FUNCTION_BLOCK EulerAngleOrientation EXTENDS AngleSequenceOrientation
VAR_INPUT
END_VAR
VAR_OUTPUT
END_VAR
VAR
	Angles_ : ARRAY [0..2] OF LREAL; 
	Sequence_ : EulerAngleSequence;
END_VAR

METHOD PUBLIC Clear
VAR_INPUT
END_VAR
Angles_[0] := 0;
Angles_[1] := 0;
Angles_[2] := 0;
END_METHOD

METHOD PUBLIC CopyFrom
VAR_INPUT
	O : EulerAngleOrientation;
END_VAR
CLEAR();
Sequence := O.Sequence;
AngleAccessor.CopyFrom(O.AngleAccessor);
END_METHOD

METHOD PUBLIC  GetAngle : LREAL
VAR_INPUT
	I : UINT;
END_VAR
VAR
	Angles : ARRAY [0..2] OF LREAL;
END_VAR
IF I >= Length THEN
	GetAngle := 0;
	RETURN;
END_IF

GetAngle := Angles[I];
END_METHOD

METHOD PUBLIC  GetDimension : Dimension
VAR_INPUT
	I : UINT;
END_VAR
VAR
	Dims : ARRAY [0..2] OF Dimension;
END_VAR
IF I >= Length THEN
	GetDimension := 0;
	RETURN;
END_IF

Dims := GetDimensions();
GetDimension := Dims[I];
END_METHOD

METHOD PUBLIC GetDimensions : ARRAY [0..2] OF Dimension
VAR_INPUT
END_VAR
CASE Sequence OF
	EulerAngleSequence.XYX:
		GetDimensions[0] := 0;
		GetDimensions[1] := 1;
		GetDimensions[2] := 0;
	EulerAngleSequence.XZX:
		GetDimensions[0] := 0;
		GetDimensions[1] := 2;
		GetDimensions[2] := 0;
	EulerAngleSequence.YXY:
		GetDimensions[0] := 1;
		GetDimensions[1] := 0;
		GetDimensions[2] := 1;
	EulerAngleSequence.YZY:
		GetDimensions[0] := 1;
		GetDimensions[1] := 2;
		GetDimensions[2] := 1;
	EulerAngleSequence.ZXZ:
		GetDimensions[0] := 2;
		GetDimensions[1] := 0;
		GetDimensions[2] := 2;
	EulerAngleSequence.ZYZ:
		GetDimensions[0] := 2;
		GetDimensions[1] := 1;
		GetDimensions[2] := 2;
	ELSE
		GetDimensions[0] := 0;
		GetDimensions[1] := 0;
		GetDimensions[2] := 0;
END_CASE
END_METHOD

PROPERTY Length : UINT
GET
Length := 3;
END_GET
END_PROPERTY

PROPERTY PUBLIC RaDeg : LREAL
GET
RaDeg := 180 * Angles_[0] / PI;
END_GET
SET
Angles_[0] := PI * RaDeg / 180;
END_SET
END_PROPERTY

PROPERTY PUBLIC RaRad : LREAL
GET
RaRad := Angles_[0];
END_GET
SET
Angles_[0] := RaRad;
END_SET
END_PROPERTY

PROPERTY PUBLIC RbDeg : LREAL
GET
RbDeg := 180 * Angles_[1] / PI;
END_GET
SET
Angles_[1] := PI * RbDeg / 180;
END_SET
END_PROPERTY

PROPERTY PUBLIC RbRad : LREAL
GET
RbRad := Angles_[1];
END_GET
SET
Angles_[1] := RbRad;
END_SET
END_PROPERTY

PROPERTY PUBLIC RcDeg : LREAL
GET
RcDeg := 180 * Angles_[2] / PI;
END_GET
SET
Angles_[2] := PI * RcDeg / 180;
END_SET
END_PROPERTY

PROPERTY PUBLIC RcRad : LREAL
GET
RcRad := Angles_[2];
END_GET
SET
Angles_[2] := RcRad;
END_SET
END_PROPERTY

PROPERTY PUBLIC Sequence : EulerAngleSequence
GET
Sequence := Sequence_;
END_GET
SET
Sequence_ := Sequence;
END_SET
END_PROPERTY

METHOD PUBLIC  SetAngle : BOOL
VAR_INPUT
	I : UINT;
	Val : LREAL;
END_VAR
VAR
	Angles : ARRAY [0..2] OF LREAL;
END_VAR
IF I >= Length THEN
	GetAngle := 0;
	SetAngle := FALSE;
	RETURN;
END_IF

SetAngle := TRUE;
Angles_[I] := Val;
END_METHOD

METHOD PUBLIC SetFromComponentsDeg
VAR_INPUT
	Ra : LREAL;
	Rb : LREAL;
	Rc : LREAL;
	Seq : EulerAngleSequence;
END_VAR
RaDeg := Ra;
RbDeg := Rb;
RcDeg := Rc;
Sequence := Seq;
END_METHOD

METHOD PUBLIC SetFromComponentsRad
VAR_INPUT
	Ra : LREAL;
	Rb : LREAL;
	Rc : LREAL;
	Seq : EulerAngleSequence;
END_VAR
RaRad := Ra;
RbRad := Rb;
RcRad := Rc;
Sequence := Seq;
END_METHOD

END_FUNCTION_BLOCK

(* stored: Version 1.1.0.1, ProductVersion 3.1.4024.9
   POU EulerAngleOrientation: Id {6250414d-7ffc-0b08-01d4-0bd3302e692f}, SpecialFunc None
   Folder Getters: Id {91c868c0-17e3-03c8-3247-0f5dcd5f58b0}
   Folder Properties: Id {b3a14366-a718-0072-0ea3-e15a9f6a7faf}
   Folder Setters: Id {bf9614b6-5791-052d-36d3-a6fecf42a028}
   Method Clear: Id {9715391d-d57d-0b5c-2943-b0eac01ec440}
   Method CopyFrom: Id {75d1fa04-b22c-0221-1769-0cfaa8bde191}
   Method GetAngle: Id {58f01ac2-632f-0309-3608-db069ea93297}
   Method GetDimension: Id {82228fe6-f24f-08e0-1dc7-5be2f0c94535}
   Method GetDimensions: Id {75983734-9b8f-0a4b-2351-422179b409ea}
   Property Length: Id {b82e00c0-8a9b-03c0-2038-f6551aefcff2}
   Get Get: Id {61adad19-8228-0348-39f4-3f87acfad94f}
   Property RaDeg: Id {7590ef98-b75c-0b20-0e44-dc9b4e96d426}
   Get Get: Id {a9c17d29-747f-0af5-3fca-dd0ac5f6e9f1}
   Set Set: Id {7b341c93-38cc-076a-1f7b-e3a6d7ade0f7}
   Property RaRad: Id {b4f0f8cd-f767-01ec-270c-2546195198f1}
   Get Get: Id {c934429d-4423-0f16-3fad-baa321bd6f39}
   Set Set: Id {c9eb25df-cd0e-0de7-3f74-91af35978334}
   Property RbDeg: Id {e0727229-9a66-00a7-0932-7525874fed84}
   Get Get: Id {7e7a3c89-650d-0223-1856-c4dac77c99bd}
   Set Set: Id {d2bc4b30-2d8c-086f-0a84-a102d8a924d9}
   Property RbRad: Id {50ee624c-31c5-0f46-30f2-042a4370722e}
   Get Get: Id {e20689c3-262e-0298-0920-0e903e52c0b0}
   Set Set: Id {6374b0af-8682-0f0e-0926-83a317e7a79e}
   Property RcDeg: Id {e95ae036-8ffe-0641-224a-48dfed486881}
   Get Get: Id {a2990168-a5aa-0e91-03d0-a19e040ae232}
   Set Set: Id {62d1a790-b443-0657-3cd9-8a022febd458}
   Property RcRad: Id {c5d0d9d9-7029-0507-2dde-27c6d67e80f7}
   Get Get: Id {8d2330a4-b1da-02aa-1571-51d72b426bc1}
   Set Set: Id {73c7808d-c208-078f-3df1-80d68d8b675a}
   Property Sequence: Id {293aad27-2052-09a0-2d77-a11adb7ed64a}
   Get Get: Id {b44d5053-7e73-0e50-1a65-5b61c95a20cd}
   Set Set: Id {b1db0a32-c79e-08c4-19ca-4b3a4a909827}
   Method SetAngle: Id {ac5bdeed-6a79-0a61-1b23-9e707ff2c1a6}
   Method SetFromComponentsDeg: Id {80cd5fd9-05ce-0de9-11ff-3c929c728842}
   Method SetFromComponentsRad: Id {4688a918-e438-0ac0-0cd1-6ae1eab851fc} *)
